(* IEC 61131-3 sources: Concurso_PLC/plc/codesys/04_FB, 8 files *)

(* ---- FB_AlarmManager.st ---- *)
(* Gestor de alarmas: enclavamiento, reconocimiento con Reset y mascaras para el HMI.
   Una alarma solo se borra con Reset cuando su condicion ya desaparecio. *)
FUNCTION_BLOCK FB_AlarmManager
VAR_INPUT
    xReset         : BOOL;   (* Nivel: reconocer y borrar (usar pulso estirado ~200 ms) *)
END_VAR
VAR_IN_OUT
    aAlarm         : ARRAY[1..GVL_Param.ALARM_COUNT] OF ST_Alarm;
END_VAR
VAR_OUTPUT
    xAnyEmergency  : BOOL;
    xAnyFault      : BOOL;
    xAnyWarning    : BOOL;
    xAnyUnack      : BOOL;
    dwActiveMask   : DWORD;
    dwUnackMask    : DWORD;
    iActiveCount   : INT;
END_VAR
VAR
    i              : INT;
END_VAR

xAnyEmergency := FALSE;
xAnyFault     := FALSE;
xAnyWarning   := FALSE;
xAnyUnack     := FALSE;
dwActiveMask  := 0;
dwUnackMask   := 0;
iActiveCount  := 0;

FOR i := 1 TO GVL_Param.ALARM_COUNT DO
    (* Flanco ascendente de la condicion: nueva ocurrencia *)
    IF aAlarm[i].xCondition AND NOT aAlarm[i].xPrevCond THEN
        aAlarm[i].xActive  := TRUE;
        aAlarm[i].xUnack   := TRUE;
        aAlarm[i].udiCount := aAlarm[i].udiCount + 1;
    END_IF
    aAlarm[i].xPrevCond := aAlarm[i].xCondition;

    (* Reset: reconoce todo y borra lo que ya no tiene causa *)
    IF xReset THEN
        aAlarm[i].xUnack := FALSE;
        IF NOT aAlarm[i].xCondition THEN
            aAlarm[i].xActive := FALSE;
        END_IF
    END_IF

    IF aAlarm[i].xActive THEN
        iActiveCount := iActiveCount + 1;
        dwActiveMask := dwActiveMask OR SHL(DWORD#1, i - 1);
        CASE aAlarm[i].eClass OF
            E_AlarmClass.EMERGENCY: xAnyEmergency := TRUE;
            E_AlarmClass.FAULT:     xAnyFault     := TRUE;
            E_AlarmClass.WARNING:   xAnyWarning   := TRUE;
        END_CASE
    END_IF
    IF aAlarm[i].xUnack THEN
        xAnyUnack   := TRUE;
        dwUnackMask := dwUnackMask OR SHL(DWORD#1, i - 1);
    END_IF
END_FOR

(* ---- FB_ColorDiverter.st ---- *)
(* Segregacion por color a la salida de cada centro de mecanizado.
   La faja de salida (M6 / M8) es la de producto AZUL: las piezas azules siguen de largo.
   Un sensor de vision configurado en "Green Product Lid" (S10) o "Green Product Base" (S11)
   detecta el producto verde; tras tCenter la faja se detiene y el pusher (Y03 / Y04) lo empuja
   a la faja de producto verde (M7 / M9). *)
FUNCTION_BLOCK FB_ColorDiverter
VAR_INPUT
    xEnable      : BOOL;
    xAutoMode    : BOOL;
    xManualMode  : BOOL;
    xManPush     : BOOL;            (* Pulso: un ciclo del pusher *)
    xGreen       : BOOL;            (* S10 / S11 *)
    xFrontLimit  : BOOL;
    xBackLimit   : BOOL;
    tCenter      : TIME := T#300MS;
    tTimeout     : TIME := T#3S;
    xHoldOnPush  : BOOL := TRUE;
    xReset       : BOOL;
END_VAR
VAR_OUTPUT
    xHoldBelt    : BOOL;            (* Detener la faja de salida *)
    xPush        : BOOL;
    xDiverted    : BOOL;            (* Pulso: producto verde enviado a su faja *)
    xBusy        : BOOL;
    xHome        : BOOL;
    xErrExtend   : BOOL;
    xErrRetract  : BOOL;
    eStep        : E_PusherStep;
END_VAR
VAR
    tonCenter    : TON;
    fbPusher     : FB_Pusher;
END_VAR

tonCenter(IN := xGreen AND xAutoMode, PT := tCenter);

fbPusher(xEnable     := xEnable,
         xStart      := (xAutoMode AND tonCenter.Q) OR (xManualMode AND xManPush),
         xFrontLimit := xFrontLimit,
         xBackLimit  := xBackLimit,
         tTimeout    := tTimeout,
         xReset      := xReset);

xHoldBelt   := xAutoMode AND (tonCenter.Q OR (xHoldOnPush AND fbPusher.xBusy));
xDiverted   := fbPusher.xDone AND xAutoMode;
xPush       := fbPusher.xPush;
xBusy       := fbPusher.xBusy;
xHome       := fbPusher.xHome;
xErrExtend  := fbPusher.xErrExtend;
xErrRetract := fbPusher.xErrRetract;
eStep       := fbPusher.eStep;

(* ---- FB_Conveyor.st ---- *)
(* Faja transportadora con modo Auto/Manual, marcha por demanda y contador de horas.
   En automatico la faja solo se mueve cuando hay piezas que mover (xDemand) y sigue
   tRunOn mas para vaciar el tramo: ahorra energia y desgaste. xHold la detiene
   cuando la estacion de aguas abajo esta ocupada (acumulacion). *)
FUNCTION_BLOCK FB_Conveyor
VAR_INPUT
    xEnable      : BOOL;            (* Permisivo: sin emergencia ni falla *)
    xManualMode  : BOOL;
    xAutoMode    : BOOL;            (* AUTO_RUN o AUTO_STOP *)
    xDemand      : BOOL;            (* Hay piezas en el tramo *)
    xHold        : BOOL;            (* Retencion pedida por la estacion siguiente *)
    xManualRun   : BOOL;            (* Orden manual desde el HMI *)
    tRunOn       : TIME := T#2S;
END_VAR
VAR_OUTPUT
    xMotor       : BOOL;
    udiRunTime_s : UDINT;
END_VAR
VAR
    tofRunOn     : TOF;
    tonSecond    : TON;
END_VAR

tofRunOn(IN := xDemand, PT := tRunOn);

IF NOT xEnable THEN
    xMotor := FALSE;
ELSIF xManualMode THEN
    xMotor := xManualRun;
ELSE
    xMotor := xAutoMode AND NOT xHold AND tofRunOn.Q;
END_IF

(* Contador de segundos de marcha (mantenimiento preventivo) *)
tonSecond(IN := xMotor AND NOT tonSecond.Q, PT := T#1S);
IF tonSecond.Q THEN
    udiRunTime_s := udiRunTime_s + 1;
END_IF

(* ---- FB_FeederStation.st ---- *)
(* Estacion de alimentacion: faja alimentadora + pusher de transferencia a la faja principal.
   Instancias: faja 1 (M1, S2, Y01, crudo verde) y faja 2 (M2, S4, Y02, crudo azul).
   - La faja acerca piezas hasta que S2/S4 detecta una; tras tCenter la detiene centrada frente al pusher.
   - Con la pieza centrada (xReady) y el turno concedido por la union (xPushPermit) ejecuta un ciclo del pusher.
   - La confirmacion de llegada (S5) la vigila PLC_PRG, que es quien conoce la faja principal. *)
FUNCTION_BLOCK FB_FeederStation
VAR_INPUT
    xEnable      : BOOL;            (* Permisivo general *)
    xFeed        : BOOL;            (* AUTO_RUN: se permite acercar y transferir piezas *)
    xManualMode  : BOOL;
    xManBelt     : BOOL;            (* Manual: faja *)
    xManPush     : BOOL;            (* Manual: pulso de un ciclo del pusher *)
    xPartAtEnd   : BOOL;            (* S2 / S4 *)
    xPushPermit  : BOOL;            (* Turno concedido por la logica de union *)
    xFrontLimit  : BOOL;
    xBackLimit   : BOOL;
    tCenter      : TIME := T#400MS;
    tTimeout     : TIME := T#3S;
    xReset       : BOOL;
END_VAR
VAR_OUTPUT
    xBelt        : BOOL;            (* Salida a la faja M1 / M2 *)
    xPush        : BOOL;            (* Salida al pusher Y01 / Y02 *)
    xReady       : BOOL;            (* Pieza centrada y pusher en reposo: lista para transferir *)
    xPushStart   : BOOL;            (* Pulso: el pusher acaba de iniciar un empuje *)
    xBusy        : BOOL;
    xHome        : BOOL;
    xErrExtend   : BOOL;
    xErrRetract  : BOOL;
    eStep        : E_PusherStep;
END_VAR
VAR
    tonCenter    : TON;
    fbPusher     : FB_Pusher;
    eStepPrev    : E_PusherStep;
END_VAR

tonCenter(IN := xPartAtEnd, PT := tCenter);
xReady := tonCenter.Q AND (fbPusher.eStep = E_PusherStep.IDLE);

fbPusher(xEnable     := xEnable,
         xStart      := (xFeed AND NOT xManualMode AND xReady AND xPushPermit)
                        OR (xManualMode AND xManPush),
         xFrontLimit := xFrontLimit,
         xBackLimit  := xBackLimit,
         tTimeout    := tTimeout,
         xReset      := xReset);

xPushStart := (fbPusher.eStep = E_PusherStep.EXTEND) AND (eStepPrev <> E_PusherStep.EXTEND)
              AND NOT xManualMode;
eStepPrev  := fbPusher.eStep;

(* La faja avanza hasta tener una pieza centrada y se detiene mientras el pusher trabaja *)
IF NOT xEnable THEN
    xBelt := FALSE;
ELSIF xManualMode THEN
    xBelt := xManBelt;
ELSE
    xBelt := xFeed AND NOT tonCenter.Q AND NOT fbPusher.xBusy;
END_IF

xPush       := fbPusher.xPush;
xBusy       := fbPusher.xBusy;
xHome       := fbPusher.xHome;
xErrExtend  := fbPusher.xErrExtend;
xErrRetract := fbPusher.xErrRetract;
eStep       := fbPusher.eStep;

(* ---- FB_Kpi.st ---- *)
(* Indicadores de produccion: conteo por salida (S12 tapas azules, S13 tapas verdes,
   S14 bases azules, S15 bases verdes), productos/min (ventana movil de 60 s),
   tiempo entre productos y disponibilidad. *)
FUNCTION_BLOCK FB_Kpi
VAR_INPUT
    axExit       : ARRAY[1..4] OF BOOL;  (* Sensor de llegada a cada salida *)
    xRunning     : BOOL;                 (* Maquina en AUTO_RUN *)
    xStopped     : BOOL;                 (* Maquina en FAULT o EMERGENCY *)
    xResetCount  : BOOL;
END_VAR
VAR_OUTPUT
    audiCount    : ARRAY[1..4] OF UDINT;
    udiTotal     : UDINT;
    rPPM         : REAL;
    rPPMInst     : REAL;
    rCycle_s     : REAL;
    rAvailability: REAL := 100.0;
    udiRun_s     : UDINT;
    udiFault_s   : UDINT;
END_VAR
VAR
    artExit      : ARRAY[1..4] OF R_TRIG;
    tonTick      : TON;
    aBucket      : ARRAY[0..59] OF UINT;  (* Piezas por segundo, ultimos 60 s *)
    iBucket      : INT;
    i            : INT;
    udiSum       : UDINT;
    tNow         : TIME;
    tLastExit    : TIME;
    xHaveLast    : BOOL;
    xExit        : BOOL;
END_VAR

IF xResetCount THEN
    FOR i := 1 TO 4 DO audiCount[i] := 0; END_FOR
    FOR i := 0 TO 59 DO aBucket[i] := 0; END_FOR
    udiRun_s := 0; udiFault_s := 0;
    xHaveLast := FALSE;
    rPPMInst := 0; rCycle_s := 0;
END_IF

xExit := FALSE;
udiTotal := 0;
FOR i := 1 TO 4 DO
    artExit[i](CLK := axExit[i]);
    IF artExit[i].Q THEN
        audiCount[i] := audiCount[i] + 1;
        xExit := TRUE;
    END_IF
    udiTotal := udiTotal + audiCount[i];
END_FOR

IF xExit THEN
    aBucket[iBucket] := aBucket[iBucket] + 1;
    tNow := TIME();
    IF xHaveLast THEN
        rCycle_s := TIME_TO_REAL(tNow - tLastExit) / 1000.0;
        IF rCycle_s > 0.0 THEN
            rPPMInst := 60.0 / rCycle_s;
        END_IF
    END_IF
    tLastExit := tNow;
    xHaveLast := TRUE;
END_IF

(* Base de tiempo de 1 s *)
tonTick(IN := NOT tonTick.Q, PT := T#1S);
IF tonTick.Q THEN
    IF xRunning THEN udiRun_s := udiRun_s + 1; END_IF
    IF xStopped THEN udiFault_s := udiFault_s + 1; END_IF

    udiSum := 0;
    FOR i := 0 TO 59 DO
        udiSum := udiSum + aBucket[i];
    END_FOR
    rPPM := UDINT_TO_REAL(udiSum);

    iBucket := (iBucket + 1) MOD 60;
    aBucket[iBucket] := 0;

    IF (udiRun_s + udiFault_s) > 0 THEN
        rAvailability := 100.0 * UDINT_TO_REAL(udiRun_s) / UDINT_TO_REAL(udiRun_s + udiFault_s);
    END_IF
END_IF

IF NOT xRunning THEN
    rPPMInst := 0.0;
END_IF

(* ---- FB_MachiningCenter.st ---- *)
(* Centro de mecanizado de Factory I/O (Machining Center): convierte un crudo en tapa o base.
   Tags (docs.factoryio.com/manual/parts/stations): Start, Stop, Reset, Produce Lids (salidas);
   Is Busy, Has Error, Opened, Progress (entradas). Tapas ~6 s, bases ~3 s de mecanizado.
   Instancias: MC1 = tapas (xProduceLids = TRUE), MC2 = bases (xProduceLids = FALSE).
   - xLoaded  : el robot retiro la pieza de la bahia de entrada (flanco de bajada de S8/S9).
   - xFinished: termino el mecanizado y la pieza quedo en la bahia de salida (flanco de bajada de Is Busy).
   - rUtilization: % del tiempo en automatico que la maquina estuvo ocupada (deteccion del cuello de botella). *)
FUNCTION_BLOCK FB_MachiningCenter
VAR_INPUT
    xEnable      : BOOL;            (* Sin emergencia ni falla *)
    xRun         : BOOL;            (* Celda en automatico (AUTO_RUN / AUTO_STOP) *)
    xManualMode  : BOOL;
    xManRun      : BOOL;
    xProduceLids : BOOL;
    xBusy        : BOOL;            (* Is Busy *)
    xEntry       : BOOL;            (* S8 / S9: pieza en la bahia de entrada *)
    xReset       : BOOL;
    xResetCount  : BOOL;
END_VAR
VAR_OUTPUT
    xStart       : BOOL;
    xStop        : BOOL;
    xResetOut    : BOOL;
    xLidsOut     : BOOL;
    xLoaded      : BOOL;            (* Pulso *)
    xFinished    : BOOL;            (* Pulso *)
    udiCycles    : UDINT;
    rLastCycle_s : REAL;
    rUtilization : REAL;
END_VAR
VAR
    ftEntry      : F_TRIG;
    rtBusy       : R_TRIG;
    ftBusy       : F_TRIG;
    tBusyStart   : TIME;
    tonTick      : TON;
    udiRun_s     : UDINT;
    udiBusy_s    : UDINT;
END_VAR

xStart    := xEnable AND ((NOT xManualMode AND xRun) OR (xManualMode AND xManRun));
xStop     := NOT xEnable;          (* Emergencia o falla: robot y CNC se detienen *)
xResetOut := xReset;
xLidsOut  := xProduceLids;

ftEntry(CLK := xEntry);
rtBusy(CLK := xBusy);
ftBusy(CLK := xBusy);
xLoaded   := ftEntry.Q AND xStart;
xFinished := ftBusy.Q;

IF rtBusy.Q THEN
    tBusyStart := TIME();
END_IF
IF ftBusy.Q THEN
    udiCycles    := udiCycles + 1;
    rLastCycle_s := TIME_TO_REAL(TIME() - tBusyStart) / 1000.0;
END_IF

IF xResetCount THEN
    udiRun_s := 0;
    udiBusy_s := 0;
    rUtilization := 0.0;
END_IF
tonTick(IN := NOT tonTick.Q, PT := T#1S);
IF tonTick.Q AND xRun AND xEnable THEN
    udiRun_s := udiRun_s + 1;
    IF xBusy THEN
        udiBusy_s := udiBusy_s + 1;
    END_IF
    rUtilization := 100.0 * UDINT_TO_REAL(udiBusy_s) / UDINT_TO_REAL(udiRun_s);
END_IF

(* ---- FB_Pusher.st ---- *)
(* Empujador de simple efecto con vigilancia de finales de carrera.
   Un flanco en xStart ejecuta un ciclo completo: extender -> retraer.
   Si un final de carrera no llega a tiempo -> ERROR (requiere xReset). *)
FUNCTION_BLOCK FB_Pusher
VAR_INPUT
    xEnable      : BOOL;
    xStart       : BOOL;          (* Flanco ascendente inicia el ciclo *)
    xFrontLimit  : BOOL;
    xBackLimit   : BOOL;
    tTimeout     : TIME := T#3S;
    xReset       : BOOL;
END_VAR
VAR_OUTPUT
    xPush        : BOOL;          (* Salida al actuador *)
    xBusy        : BOOL;
    xDone        : BOOL;          (* Pulso de un ciclo al terminar *)
    xErrExtend   : BOOL;
    xErrRetract  : BOOL;
    xHome        : BOOL;          (* Retraido y en reposo *)
    eStep        : E_PusherStep;
    udiCycles    : UDINT;
END_VAR
VAR
    rtStart      : R_TRIG;
    tonWatch     : TON;
    eStepPrev    : E_PusherStep;
END_VAR

rtStart(CLK := xStart);
xDone := FALSE;

(* El temporizador se reinicia automaticamente en cada cambio de paso *)
tonWatch(IN := (eStep = eStepPrev) AND
               ((eStep = E_PusherStep.EXTEND) OR (eStep = E_PusherStep.RETRACT)),
         PT := tTimeout);
eStepPrev := eStep;

(* Perdida de permisivo: retraer y abortar el ciclo (el llamador reintenta) *)
IF NOT xEnable AND ((eStep = E_PusherStep.EXTEND) OR (eStep = E_PusherStep.RETRACT)) THEN
    eStep := E_PusherStep.IDLE;
END_IF

CASE eStep OF
    E_PusherStep.IDLE:
        xPush := FALSE;
        IF rtStart.Q AND xEnable THEN
            eStep := E_PusherStep.EXTEND;
        END_IF

    E_PusherStep.EXTEND:
        xPush := TRUE;
        IF xFrontLimit THEN
            eStep := E_PusherStep.RETRACT;
        ELSIF tonWatch.Q THEN
            xErrExtend := TRUE;
            eStep := E_PusherStep.ERROR;
        END_IF

    E_PusherStep.RETRACT:
        xPush := FALSE;
        IF xBackLimit THEN
            eStep := E_PusherStep.DONE;
        ELSIF tonWatch.Q THEN
            xErrRetract := TRUE;
            eStep := E_PusherStep.ERROR;
        END_IF

    E_PusherStep.DONE:
        xPush := FALSE;
        xDone := TRUE;
        udiCycles := udiCycles + 1;
        eStep := E_PusherStep.IDLE;

    E_PusherStep.ERROR:
        xPush := FALSE;   (* Posicion segura: retraido *)
        IF xReset THEN
            xErrExtend  := FALSE;
            xErrRetract := FALSE;
            eStep := E_PusherStep.IDLE;
        END_IF
END_CASE

xBusy := (eStep = E_PusherStep.EXTEND) OR (eStep = E_PusherStep.RETRACT);
xHome := (eStep = E_PusherStep.IDLE) AND xBackLimit AND NOT xPush;

(* ---- FB_WheelSorter.st ---- *)
(* Wheel sorter (Pop Up Wheel Sorter) con regla de alternancia por color.
   Regla del jurado: un crudo VERDE va a la rama de TAPAS si es el primer verde, o a BASES si el
   verde anterior ya fue a tapas (y asi sucesivamente). Lo mismo, de forma independiente, para AZUL.
   Secuencia:
     IDLE     : llega una pieza al punto de lectura (S6.1/S6.2). Si la rama destino tiene cupo -> PREPARE.
                Si no hay cupo, M3 se retiene con la pieza en lectura (acumulacion).
     PREPARE  : ruedas elevadas y orientadas (Left/Right). M3 espera tSettle.
     TRANSFER : M3 avanza; la pieza pasa por S7 (flanco de subida y bajada) -> DONE.
     DONE     : alterna la regla para ese color y avisa a PLC_PRG (xDone).
     ERROR    : pieza en S7 sin clasificar (no es crudo verde ni azul) o tiempo excedido. Reset. *)
FUNCTION_BLOCK FB_WheelSorter
VAR_INPUT
    xEnable       : BOOL;
    xAutoMode     : BOOL;           (* AUTO_RUN o AUTO_STOP *)
    xManualMode   : BOOL;
    xManPlus      : BOOL;
    xManLeft      : BOOL;
    xManRight     : BOOL;
    eColorAtRead  : E_Color;        (* FC_ColorFromSensors(S6.1, S6.2) *)
    xPresence     : BOOL;           (* S7 *)
    xLidsFree     : BOOL;           (* Cupo en la rama de tapas *)
    xBasesFree    : BOOL;           (* Cupo en la rama de bases *)
    xLidsOnLeft   : BOOL := TRUE;
    tSettle       : TIME := T#300MS;
    tTimeout      : TIME := T#6S;
    xReset        : BOOL;
    xResetRule    : BOOL;           (* Reinicia la alternancia: el proximo de cada color va a tapas *)
END_VAR
VAR_OUTPUT
    xPlus         : BOOL;
    xLeft         : BOOL;
    xRight        : BOOL;
    xHoldMain     : BOOL;           (* M3 debe detenerse *)
    xDone         : BOOL;           (* Pulso: pieza entregada a su rama *)
    xDiscarded    : BOOL;           (* Pulso: Reset tras pieza no identificada (el operador la retiro) *)
    eDoneColor    : E_Color;
    eDoneBranch   : E_Branch;
    eNextBranch   : E_Branch;       (* Destino previsto para la pieza en lectura *)
    xWaitingBranch: BOOL;           (* Pieza lista pero la rama destino esta llena *)
    xErrUnknown   : BOOL;
    xErrTimeout   : BOOL;
    eStep         : E_SorterStep := E_SorterStep.IDLE;
    axNextToBases : ARRAY[1..2] OF BOOL;   (* [1] verde, [2] azul. FALSE = el proximo va a tapas *)
END_VAR
VAR
    eColor        : E_Color;
    eBranch       : E_Branch;
    eStepPrev     : E_SorterStep;
    tonStep       : TON;
    rtPresence    : R_TRIG;
    ftPresence    : F_TRIG;
    ftRead        : F_TRIG;
    xPartAtRead   : BOOL;
    xSeenOnSorter : BOOL;           (* La pieza en curso ya llego a S7 *)
    xLeftRead     : BOOL;           (* La pieza en curso ya salio del punto de lectura *)
    xToLeft       : BOOL;
    xMoving       : BOOL;
END_VAR

xDone       := FALSE;
xDiscarded  := FALSE;
xPartAtRead := (eColorAtRead <> E_Color.NONE);
rtPresence(CLK := xPresence);
ftPresence(CLK := xPresence);
ftRead(CLK := xPartAtRead);

IF xResetRule THEN
    axNextToBases[1] := FALSE;
    axNextToBases[2] := FALSE;
END_IF

(* Destino previsto segun la alternancia del color leido *)
CASE eColorAtRead OF
    E_Color.GREEN:
        IF axNextToBases[1] THEN eNextBranch := E_Branch.BASES; ELSE eNextBranch := E_Branch.LIDS; END_IF
    E_Color.BLUE:
        IF axNextToBases[2] THEN eNextBranch := E_Branch.BASES; ELSE eNextBranch := E_Branch.LIDS; END_IF
ELSE
    eNextBranch := E_Branch.NONE;
END_CASE

(* Vigilancia de tiempo: se reinicia en cada cambio de paso *)
tonStep(IN := xEnable AND (eStep = eStepPrev)
              AND ((eStep = E_SorterStep.PREPARE) OR (eStep = E_SorterStep.TRANSFER)),
        PT := SEL(eStep = E_SorterStep.PREPARE, tTimeout, tSettle));
eStepPrev := eStep;

IF xManualMode THEN
    (* En manual el operador mueve el sorter; el seguimiento se vacia al volver a automatico *)
    IF eStep <> E_SorterStep.ERROR THEN
        eStep := E_SorterStep.IDLE;
    END_IF
ELSIF xEnable THEN
    CASE eStep OF
        E_SorterStep.IDLE:
            IF rtPresence.Q AND xAutoMode THEN
                xErrUnknown := TRUE;                     (* Llego al sorter sin pasar por la vision *)
                eStep := E_SorterStep.ERROR;
            ELSIF xPartAtRead AND xAutoMode THEN
                IF ((eNextBranch = E_Branch.LIDS) AND xLidsFree)
                   OR ((eNextBranch = E_Branch.BASES) AND xBasesFree) THEN
                    eColor        := eColorAtRead;
                    eBranch       := eNextBranch;
                    xSeenOnSorter := FALSE;
                    xLeftRead     := FALSE;
                    eStep         := E_SorterStep.PREPARE;
                END_IF
            END_IF

        E_SorterStep.PREPARE:
            IF tonStep.Q THEN
                eStep := E_SorterStep.TRANSFER;
            END_IF

        E_SorterStep.TRANSFER:
            IF ftRead.Q THEN
                xLeftRead := TRUE;
            END_IF
            IF rtPresence.Q THEN
                xSeenOnSorter := TRUE;
            END_IF
            IF xSeenOnSorter AND ftPresence.Q THEN
                eStep := E_SorterStep.DONE;
            ELSIF tonStep.Q THEN
                xErrTimeout := TRUE;
                eStep := E_SorterStep.ERROR;
            END_IF

        E_SorterStep.DONE:
            xDone       := TRUE;
            eDoneColor  := eColor;
            eDoneBranch := eBranch;
            axNextToBases[TO_INT(eColor)] := NOT axNextToBases[TO_INT(eColor)];
            eStep       := E_SorterStep.IDLE;

    END_CASE
END_IF

(* El Reset se atiende aunque la celda este en FAULT (sin permisivo) *)
IF (eStep = E_SorterStep.ERROR) AND xReset THEN
    xDiscarded  := xErrUnknown;
    xErrUnknown := FALSE;
    xErrTimeout := FALSE;
    eStep       := E_SorterStep.IDLE;
END_IF

(* ---------- Salidas ---------- *)
IF xLidsOnLeft THEN
    xToLeft := (eBranch = E_Branch.LIDS);
ELSE
    xToLeft := (eBranch = E_Branch.BASES);
END_IF
xMoving := xEnable AND xAutoMode
           AND ((eStep = E_SorterStep.PREPARE) OR (eStep = E_SorterStep.TRANSFER));

IF xManualMode THEN
    xPlus     := xEnable AND xManPlus;
    xLeft     := xEnable AND xManLeft;
    xRight    := xEnable AND xManRight AND NOT xManLeft;
    xHoldMain := FALSE;
ELSE
    xPlus     := xMoving;
    xLeft     := xMoving AND xToLeft;
    xRight    := xMoving AND NOT xToLeft;
    CASE eStep OF
        E_SorterStep.PREPARE, E_SorterStep.ERROR:
            xHoldMain := TRUE;
        E_SorterStep.TRANSFER:
            (* La siguiente pieza espera en lectura, pero solo cuando la pieza en curso ya esta
               sobre el sorter: antes, M3 debe seguir moviendose para entregarla *)
            xHoldMain := xSeenOnSorter AND xLeftRead AND xPartAtRead;
    ELSE
        xHoldMain := xPartAtRead;                      (* IDLE / DONE: esperar decision *)
    END_CASE
END_IF

xWaitingBranch := xAutoMode AND (eStep = E_SorterStep.IDLE) AND xPartAtRead;
